RoboDK station: Exercises3_x.rdk

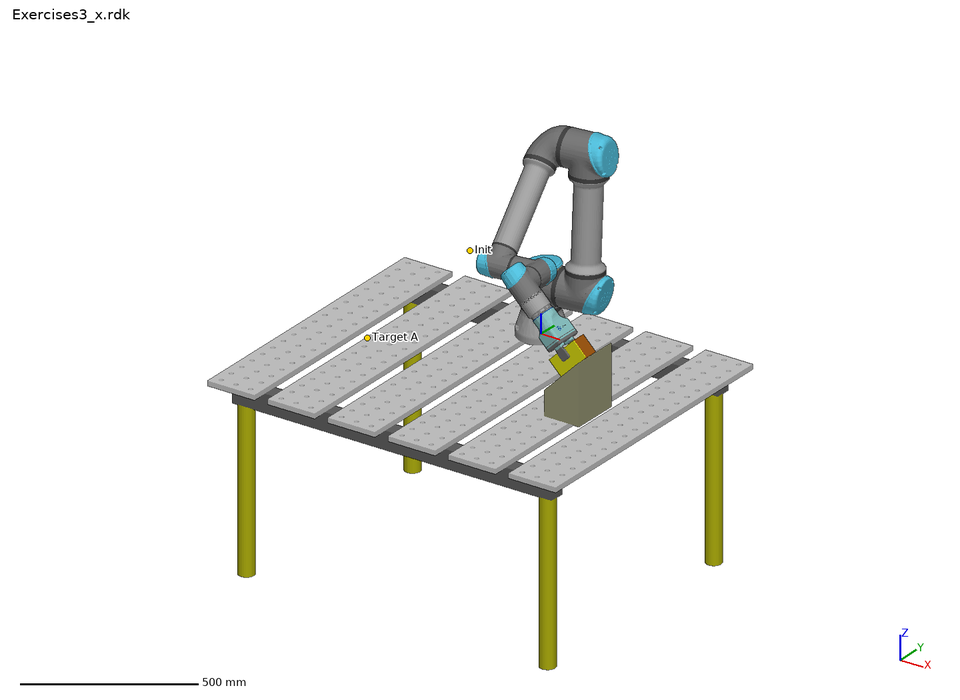
[picture v0: the station drawn from its stored meshes, robots at their saved joint values, targets as dots, program paths as lines]
Station Exercices3_x (saved by RoboDK 5.8.0). Poses are relative to the parent item; angles as X-Y-Z fixed-axis rotations.
  - frame UR5e Base at (0, 0, 0) mm
    - robot UR5e: 6 axes, payload 5 kg, reach 850 mm, repeatability 0.03 mm, weight 18.4 kg
        modified DH rows (alpha deg, a mm, theta deg, d mm): 0, 0, 0, 162.5; 90, 0, 180, 0; 0, 425, 0, 0; 0, 392.25, 0, 133.3; -90, 0, 0, 99.7; 90, 0, 180, 99.6
        joint limits [-360, -360, -360, -360, -360, -360] to [360, 360, 360, 360, 360, 360]; home [0, -90, -90, 0, 90, 0]; saved at [96.746, -94.044, 134.343, -136.999, -45.395, -260.504]
      - tool 2FG7, TCP at (0, 0, 147) mm, size 90 x 74.9 x 156.3 mm
        - object myBrick at (0, 0, 0) mm, rotated rx 180 ry 0 rz 0 deg, size 48 x 119.2 x 60.1 mm
    - target Init (joint target) at (0, -350, 400) mm, rotated rx -180 ry 0 rz 0 deg; joints [67.613, -111.82, 98.623, -76.803, -90, -202.387] of UR5e
    - target Target A (Cartesian target) at (-350, -350, 30) mm, rotated rx 180 ry 0 rz 0 deg; joints [29.377, -73.929, 122.542, -138.613, -90, -240.623] of UR5e
    - object Table at (0, 0, 0) mm, size 1193.8 x 965.2 x 609.6 mm, geometry from welding_table.sld
    - object shelf at (350, -350, 100) mm, size 120.1 x 160 x 197.5 mm, geometry from shelf.dae
    - object shelf30 at (350, -400, 100) mm, size 120.1 x 160 x 195.8 mm, geometry from shelf30.dae
    - object shelf45 at (370, -350, 100) mm, size 120.1 x 160 x 197.5 mm, geometry from shelf45.dae
